(* IEC 61131-3 sources: JaccoSigma/tempclass/Class/_XMLReader (part 2) *)

      _strcpy(hptr^.pNext^.Name, pName);
      hptr^.pNext^.pPrevious := hptr;
      hptr^.pNext^.isClosed := TRUE;

      retcode := hptr^.pNext;

    else
      // destination-element has no child -> just add
      hptr := pDest;

      hptr^.pChildren$^void := StdLib.Malloc(sizeof(_XML_ELEMENT));
      if hptr^.pChildren = NIL then
        XmlState := _ERROR;
        return;
      end_if;
      _memset(hptr^.pChildren, 0, sizeof(_XML_ELEMENT));

      NameLen := _strlen(pName) + 1;
      hptr^.pChildren^.Name$^void := StdLib.Malloc(NameLen);

      if (hptr^.pChildren^.Name = NIL) then
        XmlState := _ERROR;
        return;
      end_if;
      _strcpy(hptr^.pChildren^.Name, pName);
      hptr^.pChildren^.pFather := hptr;
      hptr^.pChildren^.isClosed := TRUE;

      retcode := hptr^.pChildren;

    end_if;
  end_if;

END_FUNCTION //AddChildElementAscii

FUNCTION _XMLReader::AddChildElementUni
	VAR_INPUT
		pDest 	: ^_XML_ELEMENT;
		pName 	: ^UINT;
	END_VAR
	VAR_OUTPUT
		retcode 	: ^_XML_ELEMENT;
	END_VAR
  VAR
  	hptr    : ^_XML_ELEMENT;
    NameLen : UDINT;
  END_VAR

  retcode := NIL;

  if (pDest = NIL) | (pName = NIL) then
    return;
  end_if;

  if pDest^.pText = NIL then
    if pDest^.pChildren <> NIL then
      // we go to the last child of our destination-element and will insert a new element with given name
      hptr := pDest^.pChildren;

      while hptr^.pNext <> NIL do
        hptr := hptr^.pNext;
      end_while;

      hptr^.pNext$^void := StdLib.Malloc(sizeof(_XML_ELEMENT));
      if hptr^.pNext = NIL then
        XmlState := _ERROR;
        return;
      end_if;
      _memset(hptr^.pNext, 0, sizeof(_XML_ELEMENT));

      NameLen := SigCLib.StrLen16(pName)*2 + 2;
      hptr^.pNext^.Name$^void := StdLib.Malloc(NameLen);

      if (hptr^.pNext^.Name = NIL) then
        XmlState := _ERROR;
        return;
      end_if;

      SigCLib.StrCpy16(hptr^.pNext^.Name$^UINT, pName);
      hptr^.pNext^.pPrevious := hptr;
      hptr^.pNext^.isClosed := TRUE;

      retcode := hptr^.pNext;

    else
      // destination-element has no child -> just add
      hptr := pDest;

      hptr^.pChildren$^void := StdLib.Malloc(sizeof(_XML_ELEMENT));
      if hptr^.pChildren = NIL then
        XmlState := _ERROR;
        return;
      end_if;
      _memset(hptr^.pChildren, 0, sizeof(_XML_ELEMENT));

      NameLen := SigCLib.StrLen16(pName)*2 + 2;
      hptr^.pChildren^.Name$^void := StdLib.Malloc(NameLen);

      if (hptr^.pChildren^.Name = NIL) then
        XmlState := _ERROR;
        return;
      end_if;
      SigCLib.StrCpy16(hptr^.pChildren^.Name$^UINT, pName);
      hptr^.pChildren^.pFather := hptr;
      hptr^.pChildren^.isClosed := TRUE;

      retcode := hptr^.pChildren;

    end_if;
  end_if;

END_FUNCTION //AddChildElementUni

FUNCTION _XMLReader::AddBrotherElementAscii
	VAR_INPUT
		pDest 	: ^_XML_ELEMENT;
		pName 	: ^USINT;
	END_VAR
	VAR_OUTPUT
		retcode 	: ^_XML_ELEMENT;
	END_VAR
  VAR
  	hptr    : ^_XML_ELEMENT;
    pSave   : ^_XML_ELEMENT;
    NameLen : UDINT;
  END_VAR

  retcode := NIL;

  if (pDest = NIL) | (pName = NIL) | (pDest = xmlStruct.MajorElement) then
    // NIL-pointer or Major Element is not able to have a Brother!
    return;
  end_if;

  if pDest^.pNext <> NIL then

    pSave := pDest^.pNext;

    hptr$^void := StdLib.Malloc(sizeof(_XML_ELEMENT));
    if hptr = NIL then
      XmlState := _ERROR;
      return;
    end_if;
    _memset(hptr, 0, sizeof(_XML_ELEMENT));

    pDest^.pNext := hptr;
    hptr^.pPrevious := pDest;

    hptr^.pNext := pSave;
    pSave^.pPrevious := hptr;

    NameLen := _strlen(pName) + 1;
    hptr^.Name$^void := StdLib.Malloc(NameLen);

    if (hptr^.Name = NIL) then
      XmlState := _ERROR;
      return;
    end_if;

    _strcpy(hptr^.Name, pName);
    hptr^.isClosed := TRUE;

    retcode := hptr;

  else

    hptr$^void := StdLib.Malloc(sizeof(_XML_ELEMENT));
    if hptr = NIL then
      XmlState := _ERROR;
      return;
    end_if;
    _memset(hptr, 0, sizeof(_XML_ELEMENT));

    pDest^.pNext := hptr;
    hptr^.pPrevious := pDest;

    NameLen := _strlen(pName) + 1;
    hptr^.Name$^void := StdLib.Malloc(NameLen);

    if (hptr^.Name = NIL) then
      XmlState := _ERROR;
      return;
    end_if;

    _strcpy(hptr^.Name, pName);
    hptr^.isClosed := TRUE;

    retcode := hptr;

  end_if;

END_FUNCTION //AddBrotherElementAscii

FUNCTION _XMLReader::AddBrotherElementUni
	VAR_INPUT
		pDest 	: ^_XML_ELEMENT;
		pName 	: ^UINT;
	END_VAR
	VAR_OUTPUT
		retcode 	: ^_XML_ELEMENT;
	END_VAR
  VAR
  	hptr    : ^_XML_ELEMENT;
    pSave   : ^_XML_ELEMENT;
    NameLen : UDINT;
  END_VAR

  retcode := NIL;

  if (pDest = NIL) | (pName = NIL) | (pDest = xmlStruct.MajorElement) then
    // NIL-pointer or Major Element is not able to have a Brother!
    return;
  end_if;

  if pDest^.pNext <> NIL then

    pSave := pDest^.pNext;

    hptr$^void := StdLib.Malloc(sizeof(_XML_ELEMENT));
    if hptr = NIL then
      XmlState := _ERROR;
      return;
    end_if;
    _memset(hptr, 0, sizeof(_XML_ELEMENT));

    pDest^.pNext := hptr;
    hptr^.pPrevious := pDest;

    hptr^.pNext := pSave;
    pSave^.pPrevious := hptr;

    NameLen := SigCLib.StrLen16(pName)*2 + 2;
    hptr^.Name$^void := StdLib.Malloc(NameLen);

    if (hptr^.Name = NIL) then
      XmlState := _ERROR;
      return;
    end_if;

    SigCLib.StrCpy16(hptr^.Name$^UINT, pName);
    hptr^.isClosed := TRUE;

    retcode := hptr;

  else

    hptr$^void := StdLib.Malloc(sizeof(_XML_ELEMENT));
    if hptr = NIL then
      XmlState := _ERROR;
      return;
    end_if;
    _memset(hptr, 0, sizeof(_XML_ELEMENT));

    pDest^.pNext := hptr;
    hptr^.pPrevious := pDest;

    NameLen := SigCLib.StrLen16(pName)*2 + 2;
    hptr^.Name$^void := StdLib.Malloc(NameLen);

    if (hptr^.Name = NIL) then
      XmlState := _ERROR;
      return;
    end_if;

    SigCLib.StrCpy16(hptr^.Name$^UINT, pName);
    hptr^.isClosed := TRUE;

    retcode := hptr;

  end_if;

END_FUNCTION //AddBrotherElementUni

FUNCTION _XMLReader::AddAttributeAscii
	VAR_INPUT
		pDest 	: ^_XML_ELEMENT;
		pName 	: ^USINT;
		pValue 	: ^USINT;
	END_VAR
	VAR_OUTPUT
		retcode 	: DINT;
	END_VAR
  VAR
  	oldSize   : UDINT;
    newSize   : UDINT;
    hptr      : ^_XML_ATTRIBUTE;
    NameLen   : UDINT;
    ValueLen  : UDINT;
  END_VAR

  retcode := -1;

  if (pDest = NIL) | (pName = NIL) | (pValue = NIL) then
    return;
  end_if;

  if pDest^.Attributes.no = 0 then
    // no attribute until now
    pDest^.Attributes.pList$^void := StdLib.Malloc(sizeof(_XML_ATTRIBUTE));
    if pDest^.Attributes.pList = NIL then
      XmlState := _ERROR;
      retcode := -2;
      return;
    end_if;

    hptr := pDest^.Attributes.pList;

    NameLen := _strlen(pName) + 1;
    ValueLen := _strlen(pValue) + 1;

    hptr^.Name$^void := StdLib.Malloc(NameLen);
    hptr^.Value$^void := StdLib.Malloc(ValueLen);

    if (hptr^.Name = NIL) | (hptr^.Value = NIL) then
      XmlState := _ERROR;
      retcode := -2;
      return;
    end_if;

    _strcpy(hptr^.Name, pName);
    _strcpy(hptr^.Value, pValue);

    pDest^.Attributes.no := 1;

  else
    // we already have at least 1 attribute -> make new attrib-list
    oldSize := pDest^.Attributes.no;
    newSize := oldSize + 1;

    hptr$^void := StdLib.Malloc(newSize * sizeof(_XML_ATTRIBUTE));
    if hptr = NIL then
      XmlState := _ERROR;
      retcode := -2;
      return;
    end_if;

    _memcpy(hptr, pDest^.Attributes.pList, oldSize * sizeof(_XML_ATTRIBUTE));
    StructCreator.FreePointer(pDest^.Attributes.pList, _XML_FREE_ATTRIBUTE);

    pDest^.Attributes.pList := hptr;

    hptr += oldSize * sizeof(_XML_ATTRIBUTE);

    NameLen := _strlen(pName) + 1;
    ValueLen := _strlen(pValue) + 1;

    hptr^.Name$^void := StdLib.Malloc(NameLen);
    hptr^.Value$^void := StdLib.Malloc(ValueLen);

    if (hptr^.Name = NIL) | (hptr^.Value = NIL) then
      XmlState := _ERROR;
      retcode := -2;
      return;
    end_if;

    _strcpy(hptr^.Name, pName);
    _strcpy(hptr^.Value, pValue);

    pDest^.Attributes.no += 1;

  end_if;

  retcode := 0;

END_FUNCTION //AddAttributeAscii

FUNCTION _XMLReader::AddAttributeUni
	VAR_INPUT
		pDest 	: ^_XML_ELEMENT;
		pName 	: ^UINT;
		pValue 	: ^UINT;
	END_VAR
	VAR_OUTPUT
		retcode 	: DINT;
	END_VAR
  VAR
  	oldSize   : UDINT;
    newSize   : UDINT;
    hptr      : ^_XML_ATTRIBUTE;
    NameLen   : UDINT;
    ValueLen  : UDINT;
  END_VAR

  retcode := -1;

  if (pDest = NIL) | (pName = NIL) | (pValue = NIL) then
    return;
  end_if;

  if pDest^.Attributes.no = 0 then
    // no attribute until now
    pDest^.Attributes.pList$^void := StdLib.Malloc(sizeof(_XML_ATTRIBUTE));
    if pDest^.Attributes.pList = NIL then
      XmlState := _ERROR;
      retcode := -2;
      return;
    end_if;

    hptr := pDest^.Attributes.pList;

    NameLen := SigCLib.StrLen16(pName)*2 + 2;
    ValueLen := SigCLib.StrLen16(pValue)*2 + 2;

    hptr^.Name$^void := StdLib.Malloc(NameLen);
    hptr^.Value$^void := StdLib.Malloc(ValueLen);

    if (hptr^.Name = NIL) | (hptr^.Value = NIL) then
      XmlState := _ERROR;
      retcode := -2;
      return;
    end_if;

    SigCLib.StrCpy16(hptr^.Name$^UINT, pName);
    SigCLib.StrCpy16(hptr^.Value$^UINT, pValue);

    pDest^.Attributes.no := 1;

  else
    // we already have at least 1 attribute -> make new attrib-list
    oldSize := pDest^.Attributes.no;
    newSize := oldSize + 1;

    hptr$^void := StdLib.Malloc(newSize * sizeof(_XML_ATTRIBUTE));
    if hptr = NIL then
      XmlState := _ERROR;
      retcode := -2;
      return;
    end_if;

    _memcpy(hptr, pDest^.Attributes.pList, oldSize * sizeof(_XML_ATTRIBUTE));
    StructCreator.FreePointer(pDest^.Attributes.pList, _XML_FREE_ATTRIBUTE);

    pDest^.Attributes.pList := hptr;

    hptr += oldSize * sizeof(_XML_ATTRIBUTE);

    NameLen := SigCLib.StrLen16(pName)*2 + 2;
    ValueLen := SigCLib.StrLen16(pValue)*2 + 2;

    hptr^.Name$^void := StdLib.Malloc(NameLen);
    hptr^.Value$^void := StdLib.Malloc(ValueLen);

    if (hptr^.Name = NIL) | (hptr^.Value = NIL) then
      XmlState := _ERROR;
      retcode := -2;
      return;
    end_if;

    SigCLib.StrCpy16(hptr^.Name$^UINT, pName);
    SigCLib.StrCpy16(hptr^.Value$^UINT, pValue);

    pDest^.Attributes.no += 1;

  end_if;

  retcode := 0;

END_FUNCTION //AddAttributeUni

FUNCTION _XMLReader::AddTextAscii
	VAR_INPUT
		pDest 	: ^_XML_ELEMENT;
		pText 	: ^USINT;
	END_VAR
	VAR_OUTPUT
		retcode 	: DINT;
	END_VAR
  VAR
  	TextLen   : UDINT;
  END_VAR

  retcode := -1;

  if (pDest = NIL) | (pText = NIL) then
    return;
  end_if;

  // only allowed to add text when element has no children or already has a text
  if (pDest^.pText <> NIL) | (pDest^.pChildren <> NIL) then
    return;
  end_if;

  TextLen := _strlen(pText);
  TextLen += 1; // zero termination

  pDest^.pText$^void := StdLib.Malloc(TextLen);
  if pDest^.pText = NIL then
    XmlState := _ERROR;
    retcode := -2;
    return;
  end_if;

  _strcpy(pDest^.pText, pText);

  retcode := 0;

END_FUNCTION //AddTextAscii

FUNCTION _XMLReader::AddTextUni
	VAR_INPUT
		pDest 	: ^_XML_ELEMENT;
		pText 	: ^UINT;
	END_VAR
	VAR_OUTPUT
		retcode 	: DINT;
	END_VAR
  VAR
  	TextLen   : UDINT;
  END_VAR

  retcode := -1;

  if (pDest = NIL) | (pText = NIL) then
    return;
  end_if;

  // only allowed to add text when element has no children or already has a text
  if (pDest^.pText <> NIL) | (pDest^.pChildren <> NIL) then
    return;
  end_if;

  TextLen := SigCLib.StrLen16(pText)*2;
  TextLen += 2; // zero termination

  pDest^.pText$^void := StdLib.Malloc(TextLen);
  if pDest^.pText = NIL then
    XmlState := _ERROR;
    retcode := -2;
    return;
  end_if;

  SigCLib.StrCpy16(pDest^.pText$^UINT, pText);

  retcode := 0;

END_FUNCTION //AddTextUni

FUNCTION _XMLReader::CreateStructAscii
	VAR_INPUT
		parsedBytes 	: ^UDINT;
	END_VAR
	VAR_OUTPUT
		retcode 	: BOOL;
	END_VAR
VAR
  pRun            : ^USINT;   // pointer to go through the information we read
  pStart          : ^USINT;   // points to the start of an element-name, atrib-name, attrib-value and so on...
  signCount       : UDINT;    // counts how much signs a string has
  counter         : UDINT;    // counter how far we passed through the information
  detectedBOM     : BOOL;
  allocRet        : DINT;
  nextSign        : USINT;
  pAttribName     : ^USINT;
  pAttribValue    : ^USINT;
  bStartReplaced  : BOOL;
END_VAR

  retcode := FALSE;

  // sprdie v2.0 - get number of elements and attributes first, afterwards get memory
  FetchElementsAndAttribsAscii(#elementCount, #attribCount);
  allocRet := StructCreator.AllocPredefinedHeap(elementCount, attribCount);
  if allocRet < 0 then
    XmlState := _ERROR;
    ErrorState := _PARSE_ERR_MEMORY;
    return;
  end_if;

  // biggest work will be here
  // we have to go through the buffer and create our XML_STRUCT out of the information
  pRun := pFileBuffer;

  counter := 1;
  bStartReplaced := FALSE;

  //sprdie v1.5 - special treatment for UTF8-BOM -----
  detectedBOM := FALSE;
  if (pRun^ = 16#EF) & ((pRun+1)^ = 16#BB) & ((pRun+2)^ = 16#BF) then
    counter += 3;
    pRun += 3;
    detectedBOM := TRUE;
  end_if;
  //--------------------------------------------------

  // first handle the header
  if (pRun^ = XML_START) & ((pRun+1)^ = '?') then

    pStart := pRun;
    signCount := 0;

    while pRun^ <> XML_END do
      signCount += 1;

      counter += 1;
      pRun += 1;
    end_while;

    // now we are pointing at the end-mark, this also has to be in the header -> increase counters
    counter += 1;
    signCount += 1;

    if signCount > XML_MAX_HEADER_LENGTH then
      return;
    end_if;

    if detectedBOM = FALSE then
      xmlStruct.Header$^void := StdLib.Malloc(signCount+1);
      _memset(xmlStruct.Header, 0, signCount+1);
      _memcpy(xmlStruct.Header, pStart, signCount);
    else
      xmlStruct.Header$^void := StdLib.Malloc(signCount+1+3); //+3 because we are going to insert the BOM to the header
      _memset(xmlStruct.Header, 0, signCount+1+3);            //   so if file is edited and written we do not lose the BOM
      _memcpy(xmlStruct.Header, pFileBuffer, signCount+3);
    end_if;

    // get memory for first element and set struct for creator
    xmlStruct.MajorElement := StructCreator.GetElementMemory(); //sprdie v2.0 - no alloc needed, get memory from struct-creator
    if (xmlStruct.MajorElement = NIL) then
      XmlState := _ERROR;
      return;
    end_if;
    _memset(xmlStruct.MajorElement, 0, sizeof(_XML_ELEMENT));
    StructCreator.SetStructPtr(#xmlStruct);

  else
    // xml does not start with the header
    ErrorState := _PARSE_ERR_NO_HEADER;
    parsedBytes^ := counter;
    return;
  end_if;

  // now lets see if we find a CR or LF and no signs between except of SPACE
  counter += 1;
  pRun += 1;
  while (pRun^ <> XML_CR) & (pRun^ <> XML_LF) & (pRun^ <> XML_START) do

    if pRun^ <> XML_SPACE then
      ErrorState := _PARSE_ERR_UNEXPECTED_SIGN;
      parsedBytes^ := counter;
      return; //wrong sign
    end_if;

    counter += 1;
    pRun += 1;
  end_while;

  // Header finished -> now lets start with looking for an Element
  searchFor := _SEARCH_ELEMENT;

  // ludben v2.3: there could only be a header in the file
  if counter = fileLength then
    ErrorState := _PARSE_ERR_NO_ROOT_ELEMENT;
    parsedBytes^ := counter;
    return;
  end_if;

  while counter < fileLength do

    case searchFor of

    	_SEARCH_ELEMENT:
    	  // look for '<'
        while (pRun^ <> XML_START) & (bStartReplaced = FALSE) do

          if (pRun^ <> XML_CR) & (pRun^ <> XML_LF) & (pRun^ <> XML_SPACE) & (pRun^ <> XML_TABULATOR) then
            ErrorState := _PARSE_ERR_UNEXPECTED_SIGN;
            parsedBytes^ := counter;
            return; //wrong sign
          end_if;

          pRun += 1;
          counter += 1;
        end_while;

        bStartReplaced := FALSE;

        // now we are pointing at start-mark, but we need one increase more
        pRun += 1;
        counter += 1;

        if (pRun^ <> XML_SLASH) & (pRun^ <> XML_EXCLAMATION) then
          //START Element
          if bTextSearched = TRUE then
            ErrorState := _PARSE_ERR_UNEXPECTED_SIGN;
            parsedBytes^ := counter;
            return; //wrong sign
          end_if;

          pStart := pRun;
          signCount := 0;

          // next step is to look for Space or End-Mark
          // counter are always one behind the pointer so we do not need to decrease afterwards
          while (pRun^ <> XML_END) & (pRun^ <> XML_SPACE) & (pRun^ <> XML_SLASH) do
            signCount += 1;

            counter += 1;
            pRun += 1;
          end_while;

          // at this point we found an element,
          nextSign := pRun^;
          pRun^ := 0; // add zero termination to file
          StructCreator.AddElement(pStart, FALSE, FALSE);

          // lets see what we have to do next
          if nextSign = XML_END then

            pRun += 1;
            counter += 1;

            if (pRun^ = XML_CR) | (pRun^ = XML_LF) | (pRun^ = XML_START) | (pRun^ = XML_SPACE) then
              searchFor := _SEARCH_ELEMENT;
            else
              searchFor := _SEARCH_TEXT;
            end_if;

          elsif nextSign = XML_SLASH then
            StructCreator.CloseElement(NIL,FALSE);

            // element is closed directly -> check if next sign is END-Tag
            pRun += 1;
            counter += 1;

            if pRun^ <> XML_END then
              // no end-tag after slash -> error
              ErrorState := _PARSE_ERR_UNEXPECTED_SIGN;
              parsedBytes^ := counter;
              return; //wrong sign
            end_if;

            // set to next sign
            pRun += 1;
            counter += 1;

            searchFor := _SEARCH_ELEMENT;

          elsif nextSign = XML_SPACE then
            // in this case there can also be a closing-tag if element ist closed directly
            if (pRun+1)^ = XML_SLASH then

              StructCreator.CloseElement(NIL, FALSE);

              //                      <Element />
              //we point now to the space-----^---
              //but we need to be after end------^
              //this means +3 signs
              pRun += 3;
              counter += 3;

              searchFor := _SEARCH_ELEMENT;
            else
              searchFor := _SEARCH_ATTRIB;
            end_if;

          end_if;

        else
          if pRun^ = XML_SLASH then

            bTextSearched := FALSE;
            // CLOSE Element
            // so just go to the end of the close-element-tag and then close
            pRun += 1;
            counter += 1;

            pStart := pRun;
            signCount := 0;

            while pRun^ <> XML_END do
              signCount += 1;

              counter += 1;
              pRun += 1;
            end_while;

            pRun^ := 0;
            pRun += 1;
            counter += 1;

            retClose := StructCreator.CloseElement(pStart, FALSE);
            if retClose <> 0 then
              ErrorState := _PARSE_ERR_WRONG_SEQUENCE;
              parsedBytes^ := counter - signCount - 1;
              return; //wrong sequence of elements
            end_if;

            searchFor := _SEARCH_ELEMENT;

          else
            // check 4 comment
            if bTextSearched = TRUE then
              ErrorState := _PARSE_ERR_UNEXPECTED_SIGN;
              parsedBytes^ := counter;
              return; //wrong sign
            end_if;

            pRun += 1;
            counter += 1;
            if (pRun^ = XML_HYPHEN) & ((pRun+1)^ = XML_HYPHEN) then
              // we found '<!--' this means comment -> skip
              pRun += 2;
              counter += 2;

              while !!((pRun^ = XML_HYPHEN) & ((pRun+1)^ = XML_HYPHEN) & ((pRun+2)^ = XML_END)) do

                pRun += 1;
                counter += 1;

              end_while;
              pRun += 3; // set ptr to one ofter end-tag
              counter += 3;
              // we found the end '-->'
              // go on with searching for an element
              searchFor := _SEARCH_ELEMENT;

            end_if;

          end_if;

        end_if;

      _SEARCH_ATTRIB:

        bTextSearched := FALSE;
    	  // when we have to search 4 an attribute we know that pRun points to a Space
        // so the next sign is the start
        pRun += 1;
        counter += 1;

        pStart := pRun;
        signCount := 0;

        while pRun^ <> XML_EQUAL do

          if (pRun^ = XML_SPACE) | (pRun^ = XML_LF) | (pRun^ = XML_CR) then
            ErrorState := _PARSE_ERR_UNEXPECTED_SIGN;
            parsedBytes^ := counter;
            return; //wrong sign
          end_if;

          signCount += 1;
          counter += 1;
          pRun += 1;
        end_while;

        pAttribName := pStart;
        pRun^ := 0;

        // we got the name of the attribute now lets get the value
        if ((pRun+1)^ <> XML_QUOTMARK) & ((pRun+1)^ <> XML_APOSTROPHE) then
          ErrorState := _PARSE_ERR_UNEXPECTED_SIGN;
          parsedBytes^ := counter;
          return; // wrong sign
        end_if;

        if ((pRun+1)^ = XML_QUOTMARK) then
          bQuot := TRUE;
        else
          bQuot := FALSE;
        end_if;

        pRun += 2; // set to one after quotation-mark
        counter += 2;

        pStart := pRun;
        signCount := 0;

        while ((pRun^ <> XML_QUOTMARK) & (bQuot = TRUE)) | ((pRun^ <> XML_APOSTROPHE) & (bQuot = FALSE)) do
          signCount += 1;

          counter += 1;
          pRun += 1;
        end_while;

        pAttribValue := pStart;
        pRun^ := 0;

        // sprdie v2.1 - convert special characters ---------------
        if (DoConvert = TRUE) then
          // convert XML notation of special characters (for example &amp; -> &)
          if ConvertXmlToText(pAttribValue, pAttribValue, sizeof(CHAR)) < 0 then // use same memory because text will be less
            ErrorState := _PARSE_ERR_UNEXPECTED_SIGN;
            parsedBytes^ := counter;
            return;
          end_if;
        end_if;
        // --------------------------------------------------------

        if StructCreator.AddAttribute(pAttribName, pAttribValue, FALSE, FALSE) = -1 then
          ErrorState := _PARSE_ERR_ATTRIBUTE_TWICE;
          parsedBytes^ := counter - signCount - 1;
          return; // attribute already exists
        end_if;

        // lets see what we have to do next
        pRun += 1;
        counter += 1;

        if pRun^ = XML_END then
          // so in this case we can have Text afterwards or next thing is an element
          pRun += 1;
          counter += 1;

          if (pRun^ = XML_CR) | (pRun^ = XML_LF) | (pRun^ = XML_START) then
            searchFor := _SEARCH_ELEMENT;
          else
            searchFor := _SEARCH_TEXT;
          end_if;

        elsif pRun^ = XML_SLASH then
            StructCreator.CloseElement(NIL, FALSE);

            // jump one sign after "/>"
            pRun += 2;
            counter += 2;
            searchFor := _SEARCH_ELEMENT;

        elsif pRun^ = XML_SPACE then
          // in this case there can also be a closing-tag if element ist closed directly
          if (pRun+1)^ = XML_SLASH then

            StructCreator.CloseElement(NIL, FALSE);

            //                      <Element />
            //we point now to the space-----^---
            //but we need to be after end------^
            //this means +3 signs
            pRun += 3;
            counter += 3;

            searchFor := _SEARCH_ELEMENT;
          else
            searchFor := _SEARCH_ATTRIB;
          end_if;

        end_if;

      _SEARCH_TEXT:
        // we already point to the start of the text
        pStart := pRun;
        signCount := 0;

        while pRun^ <> XML_START do
          signCount += 1;

          counter += 1;
          pRun += 1;
        end_while;

        // kick off text & add to actual element
        pRun^ := 0;
        bStartReplaced := TRUE;

        // sprdie v2.1 - convert special characters ---------------
        if (DoConvert = TRUE) then
          // convert XML notation of special characters (for example &amp; -> &)
          if ConvertXmlToText(pStart, pStart, sizeof(CHAR)) < 0 then // use same memory because text will be less
            ErrorState := _PARSE_ERR_UNEXPECTED_SIGN;
            parsedBytes^ := counter;
            return;
          end_if;
        end_if;
        // --------------------------------------------------------

        StructCreator.AddText(pStart, FALSE, FALSE);

        //next step has to be looking for an element
        bTextSearched := TRUE;
        searchFor := _SEARCH_ELEMENT;

    end_case;

  end_while;

  retcode := TRUE;

END_FUNCTION //CreateStructAscii

FUNCTION _XMLReader::CreateStructUni
	VAR_INPUT
		parsedBytes 	: ^UDINT;
	END_VAR
	VAR_OUTPUT
		retcode 	: BOOL;
	END_VAR
  VAR
    pRun            : ^USINT;   // pointer to go through the information we read
    pStart          : ^USINT;   // points to the start of an element-name, atrib-name, attrib-value and so on...
    signCount       : UDINT;    // counts how much signs a string has
    counter         : UDINT;    // counter how far we passed through the information
    allocRet        : DINT;
    nextSign        : UINT;
    pAttribName     : ^USINT;
    pAttribValue    : ^USINT;
    bStartReplaced  : BOOL;
  END_VAR

  retcode := FALSE;

  // sprdie v2.0 - get number of elements and attributes first, afterwards get memory
  FetchElementsAndAttribsUni(#elementCount, #attribCount);
  allocRet := StructCreator.AllocPredefinedHeap(elementCount, attribCount);
  if allocRet < 0 then
    XmlState := _ERROR;
    ErrorState := _PARSE_ERR_MEMORY;
    return;
  end_if;

  // biggest work will be here
  // we have to go through the buffer and create our XML_STRUCT out of the information
  pRun := pFileBuffer + 2;

  counter := 2;
  bStartReplaced := FALSE;

  // first handle the header
  if (pRun^$UINT = XML_START_UNI) & ((pRun+2)^$UINT = 16#003F) then

    pStart := pRun;
    signCount := 0;

    while pRun^$UINT <> XML_END_UNI do
      signCount += 2;

      counter += 2;
      pRun += 2;
    end_while;

    // now we are pointing at the end-mark, this also has to be in the header -> increase counters
    counter += 2;
    signCount += 2;

    if signCount > XML_MAX_HEADER_LENGTH then
      return;
    end_if;

    xmlStruct.Header$^void := StdLib.Malloc(signCount+2);
    _memset(xmlStruct.Header, 0, signCount+2);
    _memcpy(xmlStruct.Header, pStart, signCount);

    // alloc memory for first element and set struct for creator
    xmlStruct.MajorElement$^void := StructCreator.GetElementMemory();
    if (xmlStruct.MajorElement = NIL) then
      XmlState := _ERROR;
      return;
    end_if;
    StructCreator.SetStructPtr(#xmlStruct);

  else
    // xml does not start with the header
    ErrorState := _PARSE_ERR_NO_HEADER;
    parsedBytes^ := counter;
    return;
  end_if;

  // now lets see if we find a CR or LF and no signs between except of SPACE
  counter += 2;
  pRun += 2;
  while (pRun^$UINT <> XML_CR_UNI) & (pRun^$UINT <> XML_LF_UNI) & (pRun^$UINT <> XML_START_UNI) do

    if pRun^$UINT <> XML_SPACE_UNI then
      ErrorState := _PARSE_ERR_UNEXPECTED_SIGN;
      parsedBytes^ := counter;
      return;
    end_if;

    counter += 2;
    pRun += 2;
  end_while;

  // Header finished -> now lets start with looking for an Element
  searchFor := _SEARCH_ELEMENT;

  // ludben v2.3: there could only be a header in the file
  if counter = fileLength then
    ErrorState := _PARSE_ERR_NO_ROOT_ELEMENT;
    parsedBytes^ := counter;
    return;
  end_if;

  while counter < fileLength do

    case searchFor of

    	_SEARCH_ELEMENT:
    	  // look for '<'
        while (pRun^$UINT <> XML_START_UNI) & (bStartReplaced = FALSE) do

          if (pRun^$UINT <> XML_CR_UNI) & (pRun^$UINT <> XML_LF_UNI) & (pRun^$UINT <> XML_SPACE_UNI) & (pRun^$UINT <> XML_TABULATOR_UNI) then
            ErrorState := _PARSE_ERR_UNEXPECTED_SIGN;
            parsedBytes^ := counter;
            return;
          end_if;

          pRun += 2;
          counter += 2;
        end_while;

        bStartReplaced := FALSE;

        // now we are pointing at start-mark, but we need one increase more
        pRun += 2;
        counter += 2;

        if (pRun^$UINT <> XML_SLASH_UNI) & (pRun^$UINT <> XML_EXCLAMATION_UNI) then
          //START Element
          if bTextSearched = TRUE then
            ErrorState := _PARSE_ERR_UNEXPECTED_SIGN;
            parsedBytes^ := counter;
            return;
          end_if;

          pStart := pRun;
          signCount := 0;

          // next step is to look for Space or End-Mark
          // counter are always one behind the pointer so we do not need to decrease afterwards
          while (pRun^$UINT <> XML_END_UNI) & (pRun^$UINT <> XML_SPACE_UNI) & (pRun^$UINT <> XML_SLASH_UNI) do
            signCount += 2;

            counter += 2;
            pRun += 2;
          end_while;

          // at this point we found an element and we can get the name, so kick off name and add element to struct
          nextSign := pRun^$UINT;
          pRun^ := 0;
          StructCreator.AddElement(pStart, TRUE, FALSE);

          // lets see what we have to do next
          if nextSign = XML_END_UNI then

            pRun += 2;
            counter += 2;

            if (pRun^$UINT = XML_CR_UNI) | (pRun^$UINT = XML_LF_UNI) | (pRun^$UINT = XML_START_UNI) | (pRun^$UINT = XML_SPACE_UNI) then
              searchFor := _SEARCH_ELEMENT;
            else
              searchFor := _SEARCH_TEXT;
            end_if;

          elsif nextSign = XML_SLASH_UNI then
            StructCreator.CloseElement(NIL, TRUE);

            // element is closed directly -> check if next sign is END-Tag
            pRun += 2;
            counter += 2;

            if pRun^ <> XML_END_UNI then
              // no end-tag after slash -> error
              ErrorState := _PARSE_ERR_UNEXPECTED_SIGN;
              parsedBytes^ := counter;
              return;
            end_if;

            // set to next sign
            pRun += 2;
            counter += 2;

            searchFor := _SEARCH_ELEMENT;

          elsif nextSign = XML_SPACE_UNI then
            // in this case there can also be a closing-tag if element ist closed directly
            if (pRun+2)^ = XML_SLASH_UNI then

              StructCreator.CloseElement(NIL, TRUE);

              //                      <Element />
              //we point now to the space-----^---
              //but we need to be after end------^
              //this means +3 signs (in case of unicode 6Bytes)
              pRun += 6;
              counter += 6;

              searchFor := _SEARCH_ELEMENT;
            else
              searchFor := _SEARCH_ATTRIB;
            end_if;
          end_if;

        else
          if pRun^$UINT = XML_SLASH_UNI then

            bTextSearched := FALSE;
            // CLOSE Element
            // so just go to the end of the close-element-tag and then close
            pRun += 2;
            counter += 2;

            pStart := pRun;
            signCount := 0;

            while pRun^$UINT <> XML_END_UNI do
              signCount += 2;

              counter += 2;
              pRun += 2;
            end_while;

            pRun^ := 0;
            pRun += 2;
            counter += 2;

            retClose := StructCreator.CloseElement(pStart, TRUE);
            if retClose <> 0 then
              ErrorState := _PARSE_ERR_WRONG_SEQUENCE;
              parsedBytes^ := counter - signCount - 2;
              return;
            end_if;

            searchFor := _SEARCH_ELEMENT;

          else
            // check 4 comment
            if bTextSearched = TRUE then
              ErrorState := _PARSE_ERR_UNEXPECTED_SIGN;
              parsedBytes^ := counter;
              return;
            end_if;

            pRun += 2;
            counter += 2;
            if (pRun^$UINT = XML_HYPHEN_UNI) & ((pRun+2)^$UINT = XML_HYPHEN_UNI) then
              // we found '<!--' this means comment -> skip
              pRun += 4;
              counter += 4;

              while !!((pRun^$UINT = XML_HYPHEN_UNI) & ((pRun+2)^$UINT = XML_HYPHEN_UNI) & ((pRun+4)^$UINT = XML_END_UNI)) do

                pRun += 2;
                counter += 2;

              end_while;
              pRun += 6; // set ptr to one ofter end-tag
              counter += 6;
              // we found the end '-->'
              // go on with searching for an element
              searchFor := _SEARCH_ELEMENT;

            end_if;

          end_if;

        end_if;

      _SEARCH_ATTRIB:

        bTextSearched := FALSE;
    	  // when we have to search 4 an attribute we know that pRun points to a Space
        // so the next sign is the start
        pRun += 2;
        counter += 2;

        pStart := pRun;
        signCount := 0;

        while pRun^$UINT <> XML_EQUAL_UNI do

          if (pRun^$UINT = XML_SPACE_UNI) | (pRun^$UINT = XML_LF_UNI) | (pRun^$UINT = XML_CR_UNI) then
            ErrorState := _PARSE_ERR_UNEXPECTED_SIGN;
            parsedBytes^ := counter;
            return;
          end_if;

          signCount += 2;
          counter += 2;
          pRun += 2;
        end_while;

        pAttribName := pStart;
        pRun^ := 0;

        // we got the name of the attribute now lets get the value
        if ((pRun+2)^$UINT <> XML_QUOTMARK_UNI) & ((pRun+2)^$UINT <> XML_APOSTROPHE_UNI) then
          ErrorState := _PARSE_ERR_UNEXPECTED_SIGN;
          parsedBytes^ := counter;
          return;
        end_if;

        if ((pRun+2)^$UINT = XML_QUOTMARK_UNI) then
          bQuot := TRUE;
        else
          bQuot := FALSE;
        end_if;

        pRun += 4; // set to one after quotation-mark
        counter += 4;

        pStart := pRun;
        signCount := 0;

        while ((pRun^$UINT <> XML_QUOTMARK_UNI) & (bQuot = TRUE)) | ((pRun^$UINT <> XML_APOSTROPHE_UNI) & (bQuot = FALSE)) do
          signCount += 2;

          counter += 2;
          pRun += 2;
        end_while;

        pAttribValue := pStart;
        pRun^ := 0;

        // sprdie v2.1 - convert special characters ---------------
        if (DoConvert = TRUE) then
          // convert XML notation of special characters (for example &amp; -> &)
          if ConvertXmlToText(pAttribValue, pAttribValue, sizeof(UINT)) < 0 then // use same memory because text will be less
            ErrorState := _PARSE_ERR_UNEXPECTED_SIGN;
            parsedBytes^ := counter;
            return;
          end_if;
        end_if;
        // --------------------------------------------------------

        if StructCreator.AddAttribute(pAttribName, pAttribValue, TRUE, FALSE) = -1 then
          ErrorState := _PARSE_ERR_ATTRIBUTE_TWICE;
          parsedBytes^ := counter - signCount - 2;
          return; // attribute already exists
        end_if;

        // lets see what we have to do next
        pRun += 2;
        counter += 2;

        if pRun^$UINT = XML_END_UNI then
          // so in this case we can have Text afterwards or next thing is an element
          pRun += 2;
          counter += 2;

          if (pRun^$UINT = XML_CR_UNI) | (pRun^$UINT = XML_LF_UNI) | (pRun^$UINT = XML_START_UNI) then
            searchFor := _SEARCH_ELEMENT;
          else
            searchFor := _SEARCH_TEXT;
          end_if;

        elsif pRun^$UINT = XML_SLASH_UNI then
            StructCreator.CloseElement(NIL, TRUE);

            // jump one sign after "/>"
            pRun += 4;
            counter += 4;
            searchFor := _SEARCH_ELEMENT;

        elsif pRun^$UINT = XML_SPACE_UNI then
          // in this case there can also be a closing-tag if element ist closed directly
          if (pRun+2)^ = XML_SLASH_UNI then

            StructCreator.CloseElement(NIL, TRUE);

            //                      <Element />
            //we point now to the space-----^---
            //but we need to be after end------^
            //this means +3 signs (in case of unicode 6Bytes)
            pRun += 6;
            counter += 6;

            searchFor := _SEARCH_ELEMENT;
          else
            searchFor := _SEARCH_ATTRIB;
          end_if;

        end_if;

      _SEARCH_TEXT:
        // we already point to the start of the text
        pStart := pRun;
        signCount := 0;

        while pRun^$UINT <> XML_START_UNI do
          signCount += 2;

          counter += 2;
          pRun += 2;
        end_while;

        // kick off text & add to actual element
        pRun^ := 0;
        bStartReplaced := TRUE;

        // sprdie v2.1 - convert special characters ---------------
        if (DoConvert = TRUE) then
          // convert XML notation of special characters (for example &amp; -> &)
          if ConvertXmlToText(pStart, pStart, sizeof(UINT)) < 0 then // use same memory because text will be less
            ErrorState := _PARSE_ERR_UNEXPECTED_SIGN;
            parsedBytes^ := counter;
            return;
          end_if;
        end_if;
        // --------------------------------------------------------

        StructCreator.AddText(pStart, TRUE, FALSE);

        //next step hast to be looking for an element
        bTextSearched := TRUE;
        searchFor := _SEARCH_ELEMENT;

    end_case;

  end_while;

  retcode := TRUE;

END_FUNCTION //CreateStructUni

FUNCTION _XMLReader::FindError
	VAR_INPUT
		bytesParsed 	: UDINT;
	END_VAR
  VAR
  	count : UDINT;
    linecount : UDINT;
    signsUntilCRLF : UDINT;
    pTmp  : ^USINT;
  END_VAR

  lineCount := 1;
  signsUntilCRLF := 0;

  pTmp := pFileBuffer;

  if bRdIsUnicode = TRUE then
    pTmp += sizeof(UINT);

    bytesParsed := bytesParsed / 2;
  end_if;

  for count := 1 to bytesParsed - 1 do

    if pTmp^ = XML_LF | pTmp^ = XML_CR then
      linecount += 1;
      signsUntilCRLF := 0;

      while pTmp^ = XML_CR | pTmp^ = XML_LF do
        if bRdIsUnicode = TRUE then
          pTmp += sizeof(UINT);
        else
          pTmp += sizeof(USINT);
        end_if;
      end_while;

    else
      signsUntilCRLF += 1;

      if bRdIsUnicode = TRUE then
        pTmp += sizeof(UINT);
      else
        pTmp += sizeof(USINT);
      end_if;
    end_if;

  end_for;

  ErrorLine := TO_DINT(linecount);
  ErrorSign := TO_DINT(signsUntilCRLF);

END_FUNCTION

FUNCTION GLOBAL _XMLReader::GetAttribValueByName
	VAR_INPUT
		pElement 	: ^_XML_ELEMENT;
		pName 	: ^USINT;
	END_VAR
	VAR_OUTPUT
		pValue 	: ^USINT;
	END_VAR

  if pElement = NIL | pName = NIL then
    pValue := NIL;
    return;
  end_if;

  // look if we have tu use unicode functions or not
  if bRdIsUnicode = TRUE then
    pValue := GetAttribValueByNameUni(pElement, pName$^UINT);
  else
    pValue := GetAttribValueByNameAscii(pElement, pName);
  end_if;

END_FUNCTION

FUNCTION _XMLReader::GetAttribValueByNameAscii
	VAR_INPUT
		pElement 	: ^_XML_ELEMENT;
		pName 	: ^USINT;
	END_VAR
	VAR_OUTPUT
		pValue 	: ^USINT;
	END_VAR
  VAR
  	i : UDINT;
    pAttrib : ^_XML_ATTRIBUTE;
  END_VAR

  pValue := NIL;

  // go through whole attribute list and check names
  pAttrib := pElement^.Attributes.pList;
  for i := 1 to pElement^.Attributes.no do

    if SigCLib.StrCmp(pName, pAttrib^.Name) = 0 then
      pValue := pAttrib^.Value;
      return;
    end_if;

    pAttrib += sizeof(_XML_ATTRIBUTE);
  end_for;

END_FUNCTION

FUNCTION _XMLReader::GetAttribValueByNameUni
	VAR_INPUT
		pElement 	: ^_XML_ELEMENT;
		pName 	: ^UINT;
	END_VAR
	VAR_OUTPUT
		pValue 	: ^USINT;
	END_VAR
  VAR
  	i : UDINT;
    pAttrib : ^_XML_ATTRIBUTE;
  END_VAR

  pValue := NIL;

  // go through whole attribute list and check names
  pAttrib := pElement^.Attributes.pList;
  for i := 1 to pElement^.Attributes.no do

    if SigCLib.StrCmp16(pName, pAttrib^.Name$^UINT) = 0 then
      pValue := pAttrib^.Value;
      return;
    end_if;

    pAttrib += sizeof(_XML_ATTRIBUTE);
  end_for;

END_FUNCTION

FUNCTION GLOBAL _XMLReader::GetChildByName
	VAR_INPUT
		pParent 	: ^_XML_ELEMENT;
		pName 	: ^USINT;
		number 	: UDINT;(* := 1 *)
	END_VAR
	VAR_OUTPUT
		pChild 	: ^_XML_ELEMENT;
	END_VAR

  // number = 1 means first child; number = 2 means second child and so on...
  if number = 0 then
    pChild := NIL;
    return;
  end_if;

  if pParent = NIL | pName = NIL then
    pChild := NIL;
    return;
  end_if;

  if bRdIsUnicode = TRUE then
    pChild := GetChildByNameUni(pParent, pName$^UINT, number);
  else
    pChild := GetChildByNameAscii(pParent, pName, number);
  end_if;

END_FUNCTION

FUNCTION _XMLReader::GetChildByNameAscii
	VAR_INPUT
		pParent 	: ^_XML_ELEMENT;
		pName 	: ^USINT;
		number 	: UDINT;
	END_VAR
	VAR_OUTPUT
		pChild 	: ^_XML_ELEMENT;
	END_VAR
  VAR
  	pTmp : ^_XML_ELEMENT;
    tmpNr : UDINT;
  END_VAR

  pChild := NIL;

  // set temp-pointer to first child
  pTmp := pParent^.pChildren;
  tmpNr := number;

  while pTmp <> NIL do
    // go through childs and compare names
    if SigCLib.StrCmp(pTmp^.Name, pName) = 0 then

      tmpNr -= 1;
      if tmpNr = 0 then
        pChild := pTmp;
        return;
      end_if;

    end_if;

    pTmp := pTmp^.pNext;
  end_while;

END_FUNCTION

FUNCTION _XMLReader::GetChildByNameUni
	VAR_INPUT
		pParent 	: ^_XML_ELEMENT;
		pName 	: ^UINT;
		number 	: UDINT;
	END_VAR
	VAR_OUTPUT
		pChild 	: ^_XML_ELEMENT;
	END_VAR
  VAR
  	pTmp : ^_XML_ELEMENT;
    tmpNr : UDINT;
  END_VAR

  pChild := NIL;

  // set temp-pointer to first child
  pTmp := pParent^.pChildren;
  tmpNr := number;

  while pTmp <> NIL do
    // go through childs and compare names
    if SigCLib.StrCmp16(pTmp^.Name$^UINT, pName) = 0 then

      tmpNr -= 1;
      if tmpNr = 0 then
        pChild := pTmp;
        return;
      end_if;

    end_if;

    pTmp := pTmp^.pNext;
  end_while;

END_FUNCTION

FUNCTION GLOBAL _XMLReader::ParseXML
	VAR_INPUT
		pData 	: ^USINT;
		length 	: UDINT;
	END_VAR
	VAR_OUTPUT
		retcode 	: BOOL;
	END_VAR

  retcode := FALSE;

  if XmlState = _READY then // check if reader is ready

    if length > 0 then // check given length

      pFileBuffer$^void := StdLib.Malloc(length);
      if pFileBuffer <> NIL then

        StructCreator.SetFileBufferInfo(pFileBuffer, length);

        // alloc memory was successfull - copy data
        _memcpy(pFileBuffer, pData, length);

        fileLength := length;

        XmlState := _PARSE_STREAM;
        readSSW := _CREATE_STRUCT;

        retcode := TRUE;
      end_if;

    end_if;

  end_if;

END_FUNCTION

FUNCTION GLOBAL _XMLReader::GetXmlState
	VAR_OUTPUT
		state 	: XML_READ_STATE;
	END_VAR

  state := XmlState;

END_FUNCTION

FUNCTION GLOBAL _XMLReader::GetErrorState
	VAR_OUTPUT
		state 	: _XML_PARSE_ERROR;
	END_VAR

  state := ErrorState;

END_FUNCTION

FUNCTION _XMLReader::CreateTaskName
	VAR_INPUT
		pName 	: ^CHAR;
	END_VAR
	VAR_OUTPUT
		retcode 	: BOOL;
	END_VAR
  VAR
  	udCRC32       : UDINT;
    udStrLen      : UDINT;
    szObjectName  : ARRAY [0..255] OF CHAR;
    szCRC32       : ARRAY [0..15]  OF CHAR;
  END_VAR

  retcode := FALSE;

  if pName = NIL then
    return;
  end_if;

  SigCLib.StrCpy(dst0 := pName,
                 src0 := XMLREADER_TASKNAME);

  _GetObjName(pThis := this,
              pName := #szObjectName[0]);

  udStrLen := SigCLib.StrLen(str := #szObjectName[0]);

  udCRC32  := CheckSum.CRC32(pBuffer  := #szObjectName[0],
                             len      := udStrLen,
                             CrcStart := 0);

  SigCLib.IToA(val  := udCRC32$DINT,
                 dst  := #szCRC32[0],
                 base := 0x10);

  SigCLib.StrCat(ps1 := pName,
                   ps2 := #szCRC32[0]);

  retcode := TRUE;

END_FUNCTION

FUNCTION _XMLReader::XmlReadTask
  VAR
    bytesParsed : UDINT;
  END_VAR

  while 1 do

    if doCreate = TRUE then

      doCreate := FALSE;
      if CreateStruct(#bytesParsed) then
        isCreated := TRUE;
      else
        FindError(bytesParsed);
        XmlState := _ERROR;
      end_if;

    end_if;

    if doFree = TRUE then
      doFree := FALSE;
      StructCreator.FreeStruct();
      isFree := TRUE;
    end_if;

    MultiTask.TASKDELAY(XMLREADER_TASKDELAY);

  end_while;

END_FUNCTION

FUNCTION _XMLReader::FetchElementsAndAttribsAscii
	VAR_INPUT
		pElementCount 	: ^UDINT;
		pAttribCount 	: ^UDINT;
	END_VAR
  VAR
  	pSearch         : ^CHAR;
    bytesRead       : UDINT;
    tmpElemCount    : UDINT;
    tmpAttribCount  : UDINT;
  END_VAR

  pSearch := pFileBuffer;
  bytesRead := 0;

  tmpElemCount := 0;
  tmpAttribCount := 0;

  while bytesRead < fileLength do

      // looking for start of Element - for example `<x`
      if (pSearch^ = XML_START) then
        bytesRead += 1;
        pSearch += 1;

        if (pSearch^ <> XML_SLASH) then
          tmpElemCount += 1;
        end_if;

      elsif (pSearch^ = XML_EQUAL) then
        bytesRead += 1;
        pSearch += 1;

        if ((pSearch^ = XML_APOSTROPHE) | (pSearch^ = XML_QUOTMARK)) then
          tmpAttribCount += 1;
        end_if;
      end_if;

      bytesRead += 1;
      pSearch += 1;
  end_while;

  pElementCount^ := tmpElemCount;
  pAttribCount^ := tmpAttribCount;

END_FUNCTION

FUNCTION _XMLReader::FetchElementsAndAttribsUni
	VAR_INPUT
		pElementCount 	: ^UDINT;
		pAttribCount 	: ^UDINT;
	END_VAR
  VAR
  	pSearch         : ^UINT;
    bytesRead       : UDINT;
    tmpElemCount    : UDINT;
    tmpAttribCount  : UDINT;
  END_VAR

  pSearch := pFileBuffer$^UINT;
  bytesRead := 0;

  tmpElemCount := 0;
  tmpAttribCount := 0;

  while bytesRead < fileLength do

      // looking for start of Element - for example `<x`
      if (pSearch^ = XML_START_UNI) then
        bytesRead += 2;
        pSearch += 2;

        if (pSearch^ <> XML_SLASH_UNI) then
          tmpElemCount += 2;
        end_if;

      elsif (pSearch^ = XML_EQUAL_UNI) then
        bytesRead += 2;
        pSearch += 2;

        if ((pSearch^ = XML_APOSTROPHE_UNI) | (pSearch^ = XML_QUOTMARK_UNI)) then
          tmpAttribCount += 2;
        end_if;
      end_if;

      bytesRead += 2;
      pSearch += 2;
  end_while;

  pElementCount^ := tmpElemCount;
  pAttribCount^ := tmpAttribCount;

END_FUNCTION

FUNCTION GLOBAL _XMLReader::ConvertXmlToText
	VAR_INPUT
		pDest 	: ^void;
		pSrc 	: ^void;
		size 	: UINT;
	END_VAR
	VAR_OUTPUT
		length 	: DINT;
	END_VAR

  if ((pDest = NIL) | (pSrc = NIL)) then
    length := -1;
    return;
  end_if;

  // initialise retcode with -2 (not supported char size)
  length := -2;

  if (size = 1) then
    length := ConvertXmlToTextAscii(pDest$^CHAR, pSrc$^CHAR);
  elsif (size = 2) then
    length := ConvertXmlToTextUni(pDest$^UINT, pSrc$^UINT);
  end_if;

END_FUNCTION

FUNCTION _XMLReader::ConvertXmlToTextAscii
	VAR_INPUT
		pDest 	: ^CHAR;
		pSrc 	: ^CHAR;
	END_VAR
	VAR_OUTPUT
		length 	: DINT;
	END_VAR
  VAR
  	pSearch   : ^CHAR;
    scIndex   : UDINT;
    pNewDest  : ^CHAR;
    pNewSrc   : ^CHAR;
    pInsert   : ^CHAR;
    tmpLength : DINT;
  END_VAR

  length := 0;

  // go through whole string and replace first sign we find
  // afterwards call method again with changed pSrc and pDest
  scIndex := 0;
  pSearch := pSrc;
  while ((pSearch^ <> 0)
       & (pSearch^ <> XML_AMPERSAND)) do

    scIndex += 1;
    pSearch += sizeof(CHAR);
  end_while;

  // copy part where no special characters have been found
  if (scIndex > 0) then
    SigCLib.MemMove(pDest, pSrc, scIndex);
  end_if;

  pInsert := pDest + scIndex;
  length += scIndex$DINT;

  if (pSearch^ = 0) then
    pInsert^ := 0;
    return; // end of string reached -> leave method

  elsif (_memcmp(pSearch, XML_CONVERT_AMPERSAND, XML_LENGTH_AMPERSAND) = 0) then
    // from &amp; to & ---------------------------------------
    pInsert^ := XML_AMPERSAND;

    pNewDest := pInsert + sizeof(CHAR);
    pNewSrc := pSearch + XML_LENGTH_AMPERSAND;
    // -------------------------------------------------------

  elsif (_memcmp(pSearch, XML_CONVERT_APOS, XML_LENGTH_APOS) = 0) then
    // from &apos; to ' --------------------------------------
    pInsert^ := XML_APOSTROPHE;

    pNewDest := pInsert + sizeof(CHAR);
    pNewSrc := pSearch + XML_LENGTH_APOS;
    // -------------------------------------------------------

  elsif (_memcmp(pSearch, XML_CONVERT_GREATER, XML_LENGTH_GREATER) = 0) then
    // from &gt; to > ----------------------------------------
    pInsert^ := XML_END;

    pNewDest := pInsert + sizeof(CHAR);
    pNewSrc := pSearch + XML_LENGTH_GREATER;
    // -------------------------------------------------------

  elsif (_memcmp(pSearch, XML_CONVERT_LESS, XML_LENGTH_LESS) = 0) then
    // from &lt; to < ----------------------------------------
    pInsert^ := XML_START;

    pNewDest := pInsert + sizeof(CHAR);
    pNewSrc := pSearch + XML_LENGTH_LESS;
    // -------------------------------------------------------

  elsif (_memcmp(pSearch, XML_CONVERT_QUOT, XML_LENGTH_QUOT) = 0) then
    // from &quot; to " --------------------------------------
    pInsert^ := XML_QUOTMARK;

    pNewDest := pInsert + sizeof(CHAR);
    pNewSrc := pSearch + XML_LENGTH_QUOT;
    // -------------------------------------------------------

  else
    // nothing matched -> return with error!
    length := -3;
    return;

  end_if;

  // when we reached this point, we have been able to insert the special character -> therefore increment length of String
  length += 1;

  tmpLength := ConvertXmlToTextAscii(pNewDest, pNewSrc);
  if (tmpLength < 0) then
    length := tmpLength;
    return;
  end_if;

  length += tmpLength;

END_FUNCTION

FUNCTION _XMLReader::ConvertXmlToTextUni
	VAR_INPUT
		pDest 	: ^UINT;
		pSrc 	: ^UINT;
	END_VAR
	VAR_OUTPUT
		length 	: DINT;
	END_VAR
  VAR
  	pSearch       : ^UINT;
    scIndex       : UDINT;
    pNewDest      : ^UINT;
    pNewSrc       : ^UINT;
    pInsert       : ^UINT;
    tmpLength     : DINT;
  END_VAR

  length := 0;

  // go through whole string and replace first sign we find
  // afterwards call method again with changed pSrc and pDest
  scIndex := 0;
  pSearch := pSrc;
  while ((pSearch^ <> 0)
       & (pSearch^ <> XML_AMPERSAND)) do

    scIndex += 1;
    pSearch += sizeof(UINT);
  end_while;

  // copy part where no special characters have been found
  if (scIndex > 0) then
    SigCLib.MemMove(pDest, pSrc, scIndex*sizeof(UINT));
  end_if;

  pInsert := pDest + (scIndex * sizeof(UINT));
  length += scIndex$DINT;

  if (pSearch^ = 0) then
    pInsert^ := 0;
    return; // end of string reached -> leave method

  elsif (_memcmp(pSearch, #strUniAmp[0], (XML_LENGTH_AMPERSAND*sizeof(UINT))) = 0) then
    // from &amp; to & ---------------------------------------
    pInsert^ := XML_AMPERSAND_UNI;

    pNewDest := pInsert + sizeof(UINT);
    pNewSrc := pSearch + (XML_LENGTH_AMPERSAND*sizeof(UINT));
    // -------------------------------------------------------

  elsif (_memcmp(pSearch, #strUniApos[0], (XML_LENGTH_APOS*sizeof(UINT))) = 0) then
    // from &apos; to ' --------------------------------------
    pInsert^ := XML_APOSTROPHE_UNI;

    pNewDest := pInsert + sizeof(UINT);
    pNewSrc := pSearch + (XML_LENGTH_APOS*sizeof(UINT));
    // -------------------------------------------------------

  elsif (_memcmp(pSearch, #strUniGreater[0], (XML_LENGTH_GREATER*sizeof(UINT))) = 0) then
    // from &gt; to > ----------------------------------------
    pInsert^ := XML_END_UNI;

    pNewDest := pInsert + sizeof(UINT);
    pNewSrc := pSearch + (XML_LENGTH_GREATER*sizeof(UINT));
    // -------------------------------------------------------

  elsif (_memcmp(pSearch, #strUniLess[0], (XML_LENGTH_LESS*sizeof(UINT))) = 0) then
    // from &lt; to < ----------------------------------------
    pInsert^ := XML_START_UNI;

    pNewDest := pInsert + sizeof(UINT);
    pNewSrc := pSearch + (XML_LENGTH_LESS*sizeof(UINT));
    // -------------------------------------------------------

  elsif (_memcmp(pSearch, #strUniQuot[0], (XML_LENGTH_QUOT*sizeof(UINT))) = 0) then
    // from &quot; to " --------------------------------------
    pInsert^ := XML_QUOTMARK_UNI;

    pNewDest := pInsert + sizeof(UINT);
    pNewSrc := pSearch + (XML_LENGTH_QUOT*sizeof(UINT));
    // -------------------------------------------------------

  else
    // nothing matched -> return with error!
    length := -3;
    return;

  end_if;

  // when we reached this point, we have been able to insert the special character -> therefore increment length of String
  length += 1;

  tmpLength := ConvertXmlToTextUni(pNewDest, pNewSrc);
  if (tmpLength < 0) then
    length := tmpLength;
    return;
  end_if;

  length += tmpLength;

END_FUNCTION

FUNCTION GLOBAL _XMLReader::ResetSearch

  //sprdie v2.1 - set length to 0 so next search-method starts from beginning
  lastLen := 0;
  lastLenValue := 0;

END_FUNCTION
